# EPICS autosave request: soft_iocs/galil_DMC/iocBoot/iocgalil_DMC_E01/GalilTest_18ID_DMC_E01Positions.req
$(P)1.DVAL
$(P)2.DVAL
$(P)3.DVAL
$(P)4.DVAL
$(P)5.DVAL
$(P)6.DVAL
$(P)7.DVAL
$(P)8.DVAL
